// ---- VISUs/Home_Multidis2.TcVIS
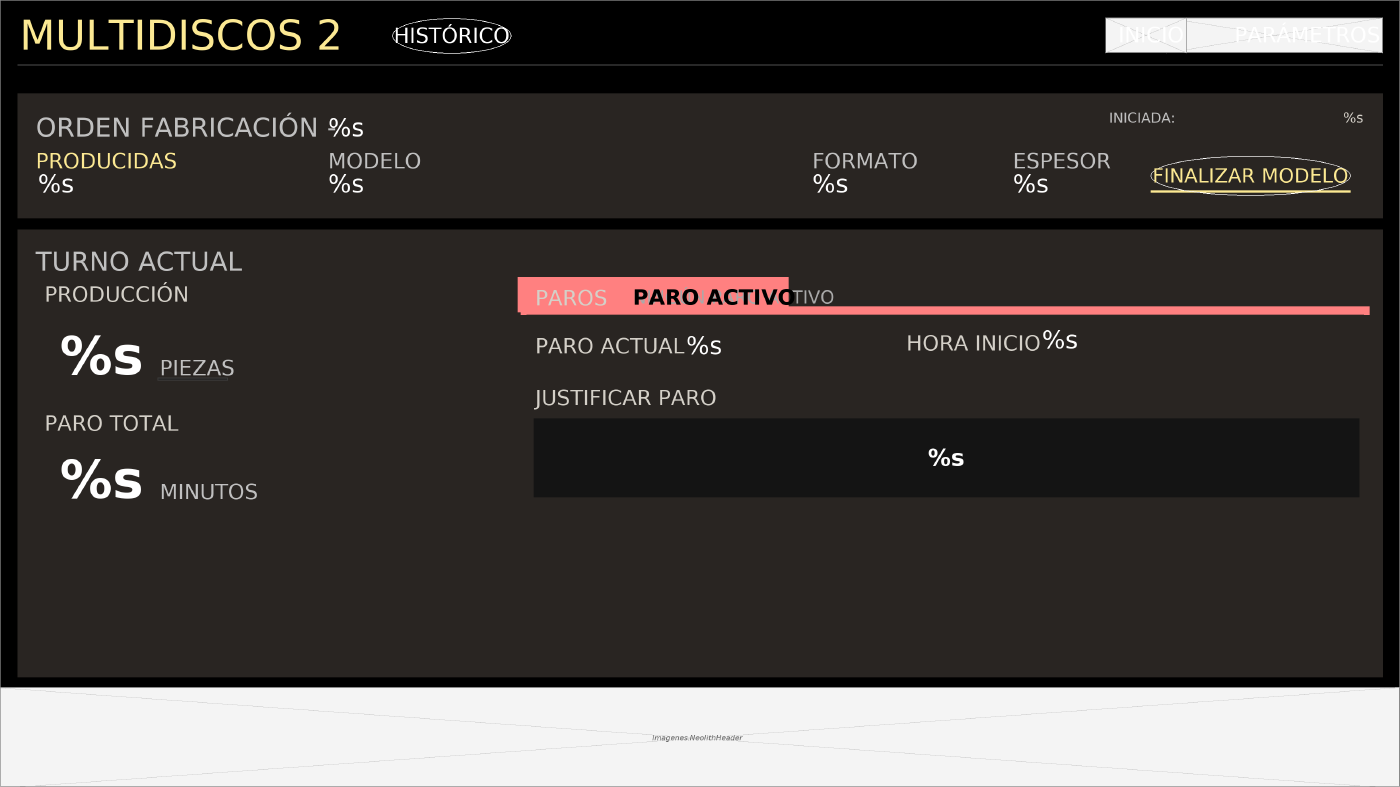
VISUALIZATION Home_Multidis2  // 1920x1080
    Ellipse (1479,1885 456x77), "Fin de producción del modelo"
        OnMouseClick: OpenDialog Dialog=V_Emerg_Fin_Prod_Md2, OpenModal=True, OpenCentered=True
    Lamp1 (869,1190 94x97), variable: FuncParoNodoMultidiscos.Funci_Multidiscos2.Fotocelula, style: Lamp-Lamp1-Yellow
    Rectangle (994,1445 183x30), "%s", text variable: FuncParoNodoCorteH4Remote1.Funci_CortHum4.H_InParo_Ftc, invisible if: FuncParoNodoMultidiscos.Funci_Multidiscos2.M_SinParo_Ftc
    Label (758,1444 239x30), "Hora Inicio del paro", invisible if: FuncParoNodoMultidiscos.Funci_Multidiscos2.M_SinParo_Ftc
    Rectangle (994,1503 192x30), "%s", text variable: FuncParoNodoCorteH4Remote1.Funci_CortHum4.Min_Parado_Ftc, invisible if: FuncParoNodoMultidiscos.Funci_Multidiscos2.M_SinParo_Ftc
    Label (793,1503 204x30), "Minutos Parado", invisible if: FuncParoNodoMultidiscos.Funci_Multidiscos2.M_SinParo_Ftc
    Label (753,1558 244x30), "Tiempo entre Piezas"
    Label (742,1594 255x62), "Tiempo entre Piezas Anterior"
    Rectangle (172,1318 183x123), "%s", text variable: FuncParoNodoMultidiscos.Funci_Multidiscos2.Cont_Piezas_Ftc
    Rectangle (994,1558 192x30), "%s", text variable: FuncParoNodoCorteH4Remote1.Funci_CortHum4.t_Entre_Piez_Ftc
    Rectangle (994,1610 192x30), "%s", text variable: FuncParoNodoCorteH4Remote1.Funci_CortHum4.t_Entr_Piez_Ante_Ftc
    Label (718,1127 397x30), "Sensor presencia tabla"
    Label (753,1348 326x30), "En producción todo OK", invisible if: FuncParoNodoMultidiscos.Funci_Multidiscos2.MParo_Ftc
    Label (571,1279 235x59), "Línea en paro", invisible if: FuncParoNodoMultidiscos.Funci_Multidiscos2.M_SinParo_Ftc
    Label (85,1180 361x144), "Número de losas"
    Label (1390,1230 361x56), "Modelo actual"
    Rectangle (1235,1324 671x53), "%s", text variable: FuncParoNodoMultidiscos.sModeloActualTabla_MD2
    Label (1390,1615 361x56), "Espesor"
    Rectangle (1235,1704 671x53), "%s", text variable: FuncParoNodoMultidiscos.sEspesorActualTabla_MD2
    Label (1390,1417 361x56), "Formato"
    Rectangle (1235,1506 671x53), "%s", text variable: FuncParoNodoMultidiscos.sFormatoActualTabla_MD2
    Rectangle (1533,1124 300x30), "%s", text variable: FuncParoNodoMultidiscos.sFechaInicModeloTab_MD2
    Label (1178,1125 354x30), "Fecha inicio del modelo actual"
    Rectangle (56,1801 1380x154), "%s", text variable: FuncParoNodoMultidiscos.Funci_Multidiscos2.S_Justi_Paro_Ftc, invisible if: FuncParoNodoMultidiscos.Funci_Multidiscos2.M_SinParo_Ftc
        OnMouseDown: write the text variable via Edit
    Label (55,1710 1381x106), "JUSTIFICAR EL PARO ACTUAL", invisible if: FuncParoNodoCorteH4Remote1.Funci_CortHum4.M_SinParo_Ftc
    Rectangle (24,315 1872x614)
    Rectangle (24,128 1872x171)
    Rectangle (24,88 1872x2)
    Label (24,16 514x64), "MULTIDISCOS 2"
    Rectangle (1426,451 183x30), "%s", text variable: FuncParoNodoCorteH4Remote1.Funci_CortHum4.H_InParo_Ftc, invisible if: FuncParoNodoMultidiscos.Funci_Multidiscos2.M_SinParo_Ftc
    Rectangle (938,459 192x30), "%s", text variable: FuncParoNodoCorteH4Remote1.Funci_CortHum4.Min_Parado_Ftc, invisible if: FuncParoNodoMultidiscos.Funci_Multidiscos2.M_SinParo_Ftc
    Label (46,148 390x54), "ORDEN FABRICACIÓN -"
    Rectangle (1573,147 300x30), "%s", text variable: FuncParoNodoMultidiscos.sFechaInicModeloTab_MD2
    Label (1518,147 99x30), "INICIADA:"
    Rectangle (732,574 1132x108), "%s", text variable: FuncParoNodoMultidiscos.Funci_Multidiscos2.S_Justi_Paro_Ftc, invisible if: FuncParoNodoMultidiscos.Funci_Multidiscos2.M_SinParo_Ftc
        OnMouseDown: write the text variable via Edit
    Image (1600,24 296x48), "PARÁMETROS"
        OnMouseClick: change screen: Ajustes_CorteH4
    Image (1516,24 111x48), "INICIO"
        OnMouseClick: change screen: Home_Sel_Maq
    Rectangle (447,232 671x40), "%s", text variable: FuncParoNodoMultidiscos.sModeloActualTabla_MD2
    Rectangle (1386,232 120x40), "%s", text variable: FuncParoNodoMultidiscos.sEspesorActualTabla_MD2
    Rectangle (1111,232 321x40), "%s", text variable: FuncParoNodoMultidiscos.sFormatoActualTabla_MD2
    Label (447,203 487x36), "MODELO"
    Label (1111,203 156x36), "FORMATO"
    Label (1386,203 156x36), "ESPESOR"
    Rectangle (447,155 321x40), "%s", text variable: FuncParoNodoCorteH4Remote1.sFormatoActualTabla
    Label (46,203 199x36), "PRODUCIDAS"
    Rectangle (49,232 248x40), "%s", text variable: FuncParoNodoCorteH4Remote1.sEspesorActualTabla
    Group (1578,214 274x54)
        Rectangle (0,47 274x3)
        Ellipse (0,0 274x54), "FINALIZAR MODELO"
            OnMouseClick: OpenDialog Dialog=V_Emerg_Fin_Prod_Md2, OpenModal=True, OpenCentered=True
    Label (46,332 390x54), "TURNO ACTUAL"
    Label (58,386 199x36), "PRODUCCIÓN"
    Label (731,457 261x36), "PARO ACTUAL", invisible if: FuncParoNodoMultidiscos.Funci_Multidiscos2.M_SinParo_Ftc
    Label (1240,453 261x36), "HORA INICIO", invisible if: FuncParoNodoMultidiscos.Funci_Multidiscos2.M_SinParo_Ftc
    Rectangle (79,444 183x88), "%s", text variable: FuncParoNodoMultidiscos.Funci_Multidiscos2.Cont_Piezas_Ftc
    Label (216,487 106x36), "PIEZAS"
    Rectangle (216,518 96x4), colour toggle: FuncParoNodoCorteH4Remote1.Funci_CortHum4.Fotocelula
    Label (731,528 261x36), "JUSTIFICAR PARO", invisible if: FuncParoNodoMultidiscos.Funci_Multidiscos2.M_SinParo_Ftc
    Rectangle (714,424 1164x4), invisible if: FuncParoNodoMultidiscos.Funci_Multidiscos2.M_SinParo_Ftc
    Rectangle (710,380 371x48), invisible if: FuncParoNodoMultidiscos.Funci_Multidiscos2.M_SinParo_Ftc
    Label (731,391 199x36), "PAROS"
    Label (865,393 326x30), "NINGÚN PARO ACTIVO", invisible if: FuncParoNodoMultidiscos.Funci_Multidiscos2.MParo_Ftc
    Label (865,393 235x30), "PARO ACTIVO", invisible if: FuncParoNodoMultidiscos.Funci_Multidiscos2.M_SinParo_Ftc
    Ellipse (538,25 163x48), "HISTÓRICO"
        OnMouseClick: change screen: HistTablaTablas_Ch4
    Label (58,563 261x36), "PARO TOTAL"
    Rectangle (79,614 183x88), "%s", text variable: FuncParoNodoCorteH4Remote1.Funci_CortHum4.Cont_Piezas_Ftc
    Label (216,657 142x36), "MINUTOS"
    Image (-7,943 1927x139), image: Imagenes.NeolithHeader
END_VISUALIZATION

// ---- VISUs/Listas_Para_Desplegables/FormatoTabla.TcTLO
TEXTLIST FormatoTabla
  0 = 'Sin seleccionar'
  1 = '170x170'
  2 = '200x650'
  3 = '300x150'
  4 = '300x300'
  5 = '30x30'
  6 = 'Ninguno de la lista'
   = ''
END_TEXTLIST

// ---- VISUs/Modelo_Tabla_Ch4.TcVIS
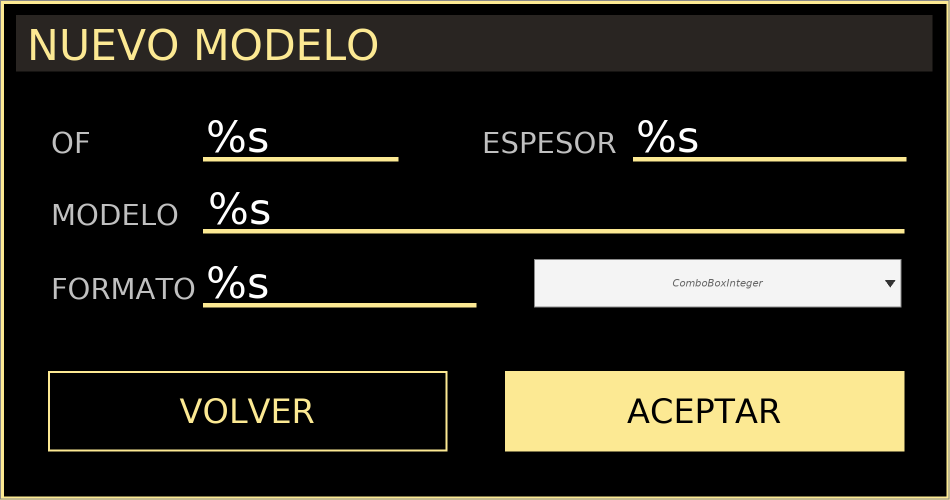
VISUALIZATION Modelo_Tabla_Ch4  // 950x500
    Rectangle (16,15 916x56)
    Rectangle (0,0 950x500)
    Label (24,17 498x56), "NUEVO MODELO"
    Rectangle (136,1125 690x58), "%s Contador piezas corte húmedo 4", text variable: FuncParoNodoCorteH4Remote1.CortHum4StrFuncParoEnviar.Cont_Piezas
    Button (871,1105 269x91), "Reset contador"
        tap FuncParoNodoCorteH4Remote1.Funci_CortHum4.ResetContPiez
    ComboBoxInteger (534,259 367x48), variable: FuncParoNodoCorteH4Remote1.FunGeneCortHum4.IndexListFormatoTabla, text list: 'FormatoTabla'
        p1601986498: ''
    Rectangle (205,185 701x48), "%s", text variable: FuncParoNodoCorteH4Remote1.FunGeneCortHum4.s_ModeloEleccionTabla
        OnMouseDown: write the text variable via Edit
    Label (48,197 148x36), "MODELO"
    Rectangle (203,229 701x4)
    Group (48,259 428x48), text variable: FuncParoNodoCorteH4Remote1.FunGeneCortHum4.s_FormatoEleccionTabla, input disabled if: FuncParoNodoCorteH4Remote1.FunGeneCortHum4.IndexListFormatoTabla<>0
        OnMouseClick: write the text variable via Edit
        Rectangle (155,0 273x48), "%s", text variable: FuncParoNodoCorteH4Remote1.sFormatoActualTabla
            OnMouseDown: write the text variable via Edit
        Label (0,12 148x36), "FORMATO"
        Rectangle (155,44 273x4)
    Group (479,113 427x48), "%s", text variable: FuncParoNodoCorteH4Remote1.FunGeneCortHum4.s_EspesorEleccionTabla
        OnMouseDown: write the text variable via Edit
        Rectangle (154,0 273x48), "%s", text variable: FuncParoNodoCorteH4Remote1.sEspesorActualTabla
            OnMouseDown: write the text variable via Edit
        Label (0,12 148x36), "ESPESOR"
        Rectangle (154,44 273x4)
    Rectangle (505,371 399x80), "ACEPTAR"
        tap FuncParoNodoCorteH4Remote1.FunGeneCortHum4.P_EscribirModelo
        OnMouseClick: CloseDialog Dialog=Modelo_Tabla_Ch4, Result=OK, NumpadKeypadSet=True
    Rectangle (48,371 399x80), "VOLVER"
        OnMouseClick: CloseDialog Dialog=Modelo_Tabla_Ch4, Result=Cancel, NumpadKeypadSet=True
    Group (48,113 350x48)
        Rectangle (155,0 195x48), "%s", text variable: FuncParoNodoCorteH4Remote1.sEspesorActualTabla
            OnMouseDown: write the text variable via Edit
        Label (0,12 148x36), "OF"
        Rectangle (155,44 195x4)
END_VISUALIZATION

// ---- VISUs/Ajustes_CorteH4.TcVIS
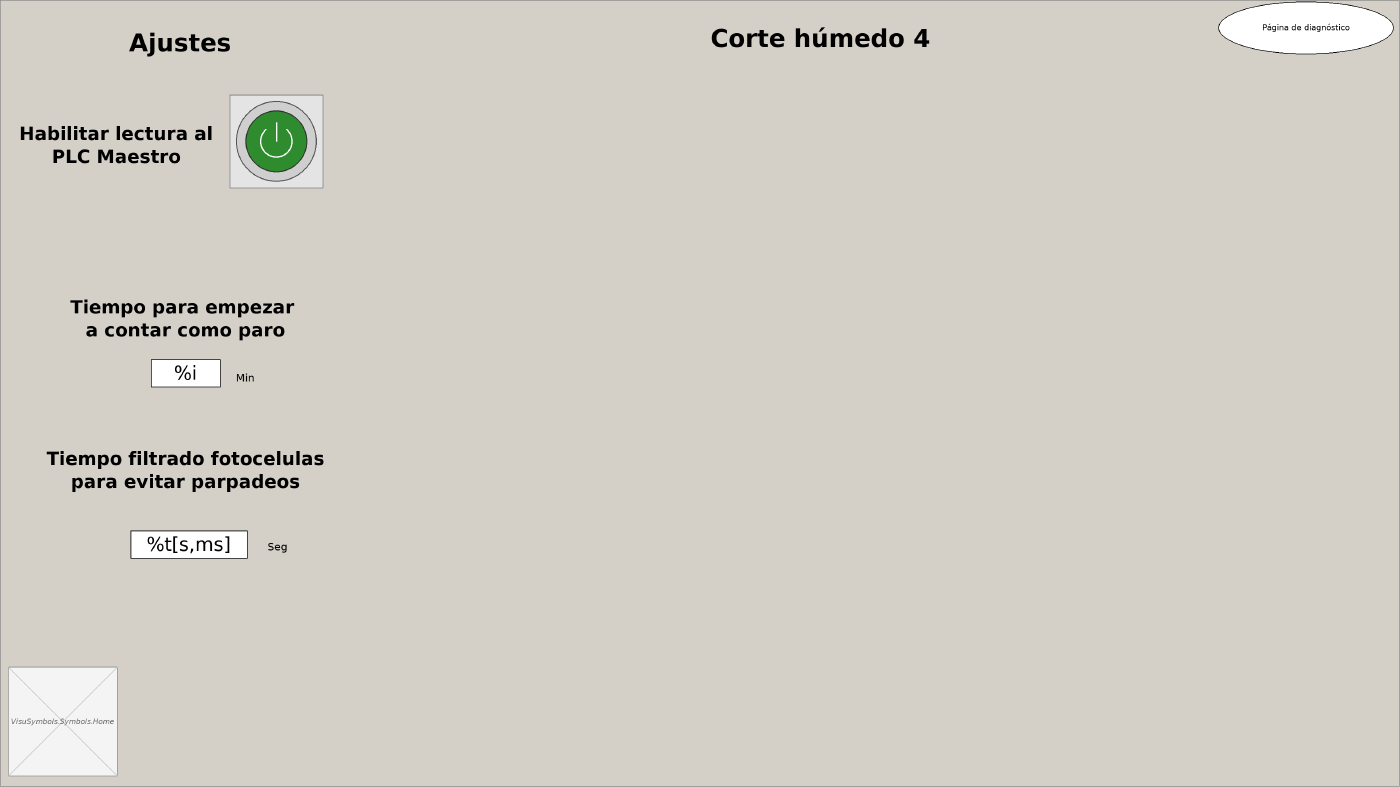
VISUALIZATION Ajustes_CorteH4  // 1920x1080
    Label (143,29 208x59), "Ajustes"
    Image (11,915 150x150), image: VisuSymbols.Symbols.Home
        OnMouseClick: change screen: Home_CortH4
    Label (22,144 275x110), "Habilitar lectura al PLC Maestro"
    PowerSwitch (315,128 128x132), variable: MAIN_Orden_Lectura_PLCs.bHabilitaLectura_Maestro, behaviour: TOGGLE, style: Switch-PowerSwitch-Green
    Label (82,390 345x94), "Tiempo para empezar a contar como paro"
    Label (160,482 188x30)
    Rectangle (207,493 95x38), "%i", text variable: FuncParoNodoCorteH4Remote1.HMI_Tiempo_Offset_MParo
        OnMouseDown: write the text variable via Edit
    Label (307,500 59x37), "Min"
    Label (58,598 393x94), "Tiempo filtrado fotocelulas para evitar parpadeos"
    Label (351,732 59x37), "Seg"
    Rectangle (179,728 160x38), "%t[s,ms]", text variable: FuncParoNodoCorteH4Remote1.HMI_TiempoFiltradoFotocel
        OnMouseDown: write the text variable via Edit
    Label (925,23 401x59), "Corte húmedo 4"
    Ellipse (1671,2 240x72), "Página de diagnóstico"
        OnMouseClick: change screen: DiagnosticoFB
END_VISUALIZATION

// ---- VISUs/Home_Sel_Maq.TcVIS
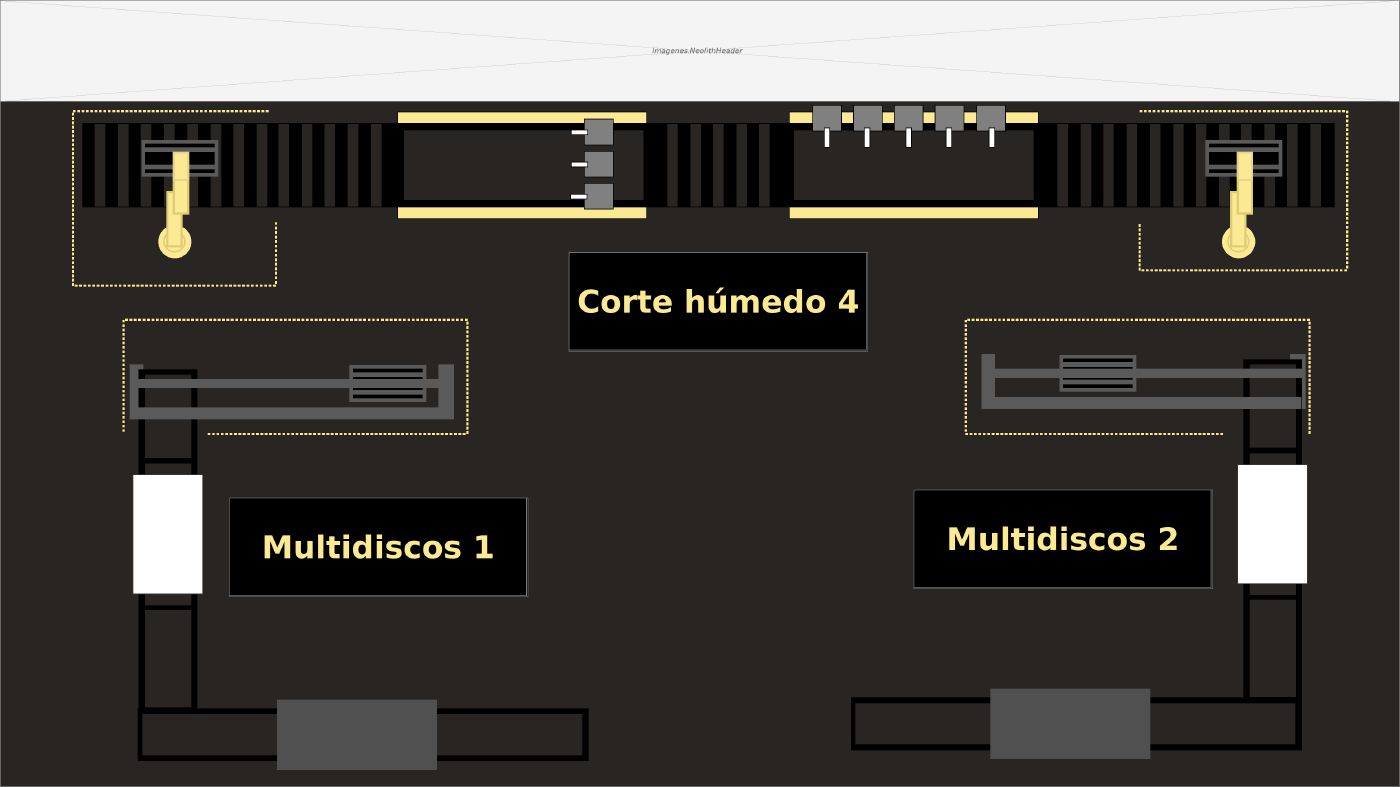
VISUALIZATION Home_Sel_Maq  // 1920x1080
    Button (780,346 410x136), "Corte húmedo 4"
        OnMouseUp: change screen: Home_CortH4
    Button (314,683 410x136), "Multidiscos 1"
        OnMouseUp: change screen: Home_Multidis1
    Button (1253,672 410x136), "Multidiscos 2"
        OnMouseDown: change screen: Home_Multidis2
    Image (-7,0 1927x139), image: Imagenes.NeolithHeader
    Group (100,144 1747x248)
        Rectangle (445,9 342x147)
        Rectangle (982,9 342x147)
        Rectangle (13,25 1717x115)
        Group (1349,25 363x115)
            Rectangle (0,0 16x115)
            Rectangle (32,0 16x115)
            Group (63,0 48x115)
                Rectangle (0,0 16x115)
                Rectangle (32,0 16x115)
            Group (127,0 111x115)
                Rectangle (0,0 16x115)
                Rectangle (32,0 16x115)
                Group (63,0 48x115)
                    Rectangle (0,0 16x115)
                    Rectangle (32,0 16x115)
            Rectangle (252,0 16x115)
            Rectangle (284,0 16x115)
            Group (315,0 48x115)
                Rectangle (0,0 16x115)
                Rectangle (32,0 16x115)
        Group (29,25 363x115)
            Rectangle (0,0 16x115)
            Rectangle (32,0 16x115)
            Group (63,0 48x115)
                Rectangle (0,0 16x115)
                Rectangle (32,0 16x115)
            Group (127,0 111x115)
                Rectangle (0,0 16x115)
                Rectangle (32,0 16x115)
                Group (63,0 48x115)
                    Rectangle (0,0 16x115)
                    Rectangle (32,0 16x115)
            Rectangle (252,0 16x115)
            Rectangle (284,0 16x115)
            Group (315,0 48x115)
                Rectangle (0,0 16x115)
                Rectangle (32,0 16x115)
        Rectangle (408,25 16x115)
        Rectangle (453,34 330x97)
        Rectangle (701,19 40x36)
        Rectangle (701,63 40x36)
        Rectangle (701,107 40x36)
        Rectangle (683,34 23x7)
        Rectangle (683,78 23x7)
        Rectangle (682,122 23x7)
        Rectangle (988,34 330x97)
        Rectangle (1014,0 40x36)
        Rectangle (1070,0 40x36)
        Rectangle (1126,0 40x36)
        Rectangle (1182,0 40x36)
        Rectangle (1239,0 40x36)
        Rectangle (1085,31 8x27)
        Rectangle (1030,31 8x27)
        Rectangle (1142,31 8x27)
        Rectangle (1197,31 8x27)
        Rectangle (1256,31 8x27)
        Group (814,25 142x115)
            Rectangle (126,0 16x115)
            Rectangle (0,0 16x115)
            Rectangle (32,0 16x115)
            Group (63,0 48x115)
                Rectangle (0,0 16x115)
                Rectangle (32,0 16x115)
        Polyline (1463,8) (1747,8) (1747,227) (1463,227) (1463,161)
        Polyline (278,161) (278,248) (0,248) (0,8) (271,8)
        Group (94,48 105x162)
            Ellipse (23,117 45x45)
            Ellipse (30,124 30x30)
            RoundedRectangle (34,70 22x77)
            RoundedRectangle (0,0 105x50)
            Rectangle (0,10 105x6)
            Rectangle (0,34 105x6)
            RoundedRectangle (43,25 22x77)
            RoundedRectangle (43,16 22x40)
        Group (1553,48 105x162)
            Ellipse (23,117 45x45)
            Ellipse (30,124 30x30)
            RoundedRectangle (34,70 22x77)
            RoundedRectangle (0,0 105x50)
            Rectangle (0,10 105x6)
            Rectangle (0,34 105x6)
            RoundedRectangle (43,25 22x77)
            RoundedRectangle (43,16 22x40)
    Group (1167,439 629x602)
        Rectangle (544,362 65x16)
        Rectangle (0,518 618x72)
        Polyline (629,156) (629,0) (157,0) (157,156) (513,156)
        Group (286,48 57x50)
            RoundedRectangle (0,0 105x50)
            Rectangle (0,10 105x6)
            Rectangle (0,34 105x6)
        Rectangle (602,47 21x75)
        Rectangle (179,47 18x75)
        Rectangle (538,54 80x465)
        Rectangle (546,60 65x116)
        Rectangle (546,182 65x196)
        Rectangle (530,198 96x164)
        Rectangle (546,383 65x135)
        Rectangle (5,525 605x58)
        Rectangle (191,506 219x96)
        Rectangle (193,106 424x16)
        Rectangle (190,67 431x12)
    Group (169,439 638x617)
        Rectangle (20,533 618x72)
        Polyline (116,156) (472,156) (472,0) (0,0) (0,156)
        Group (310,62 57x50)
            RoundedRectangle (0,0 105x50)
            Rectangle (0,10 105x6)
            Rectangle (0,34 105x6)
        Rectangle (432,61 21x75)
        Rectangle (9,61 18x75)
        Rectangle (21,68 80x465)
        Rectangle (29,74 65x116)
        Rectangle (29,196 65x196)
        Rectangle (13,212 96x164)
        Rectangle (29,397 65x135)
        Rectangle (25,540 605x58)
        Rectangle (211,521 219x96)
        Rectangle (17,120 430x16)
        Rectangle (20,81 431x12)
END_VISUALIZATION

// ---- VISUs/HistTablaTablas_Ch4.TcVIS
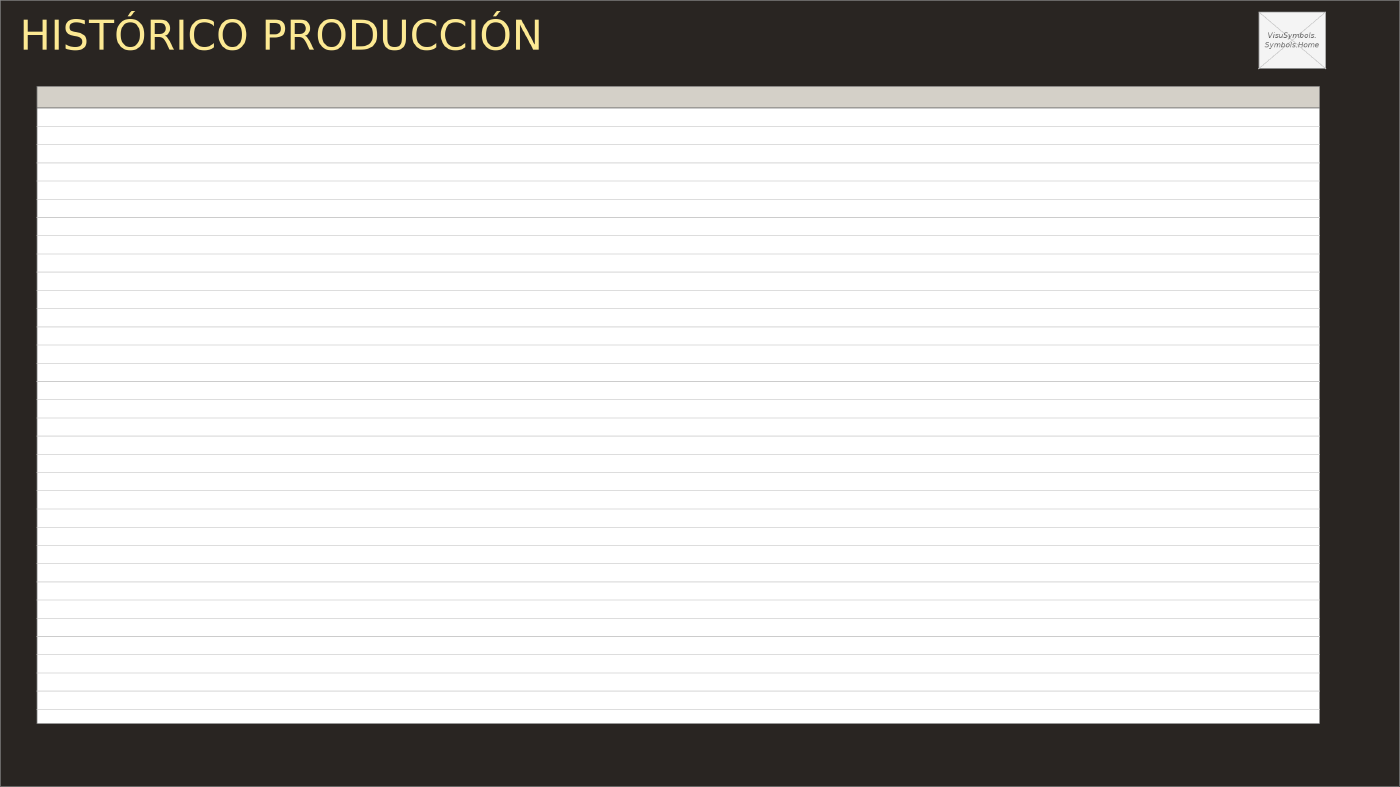
VISUALIZATION HistTablaTablas_Ch4  // 1920x1080
    Image (1726,16 92x78), image: VisuSymbols.Symbols.Home
        OnMouseClick: change screen: Home_CortH4
    Table (50,118 1760x875), data array: RegistroLocalDataBase.aHistoricStrTablasCH4
        p3854506369: RegistroLocalDataBase.aHistoricStrTablasCH4[INDEX].ID
        p1892666644: RegistroLocalDataBase.aHistoricStrTablasCH4[INDEX].Fecha
        p338671338: RegistroLocalDataBase.aHistoricStrTablasCH4[INDEX].Modelo
        p2170511999: RegistroLocalDataBase.aHistoricStrTablasCH4[INDEX].Formato
        p3723444502: RegistroLocalDataBase.aHistoricStrTablasCH4[INDEX].Espesor
        p1218418051: RegistroLocalDataBase.aHistoricStrTablasCH4[INDEX].Maquina
        p746581629: RegistroLocalDataBase.aHistoricStrTablasCH4[INDEX].Cont_Piezas
        p3104783080: RegistroLocalDataBase.aHistoricStrTablasCH4[INDEX].t_Entre_Piez_Ftc
        p2501879983: RegistroLocalDataBase.aHistoricStrTablasCH4[INDEX].S_Justi_Paro_Ftc
        p1757482276: Numero de tablas
        p4088588272: Tiempo entre tablas
        p2243050616: Justif paro
    Label (24,16 669x64), "HISTÓRICO PRODUCCIÓN"
END_VISUALIZATION

// ---- VISUs/Modelo_Tabla_Md1.TcVIS
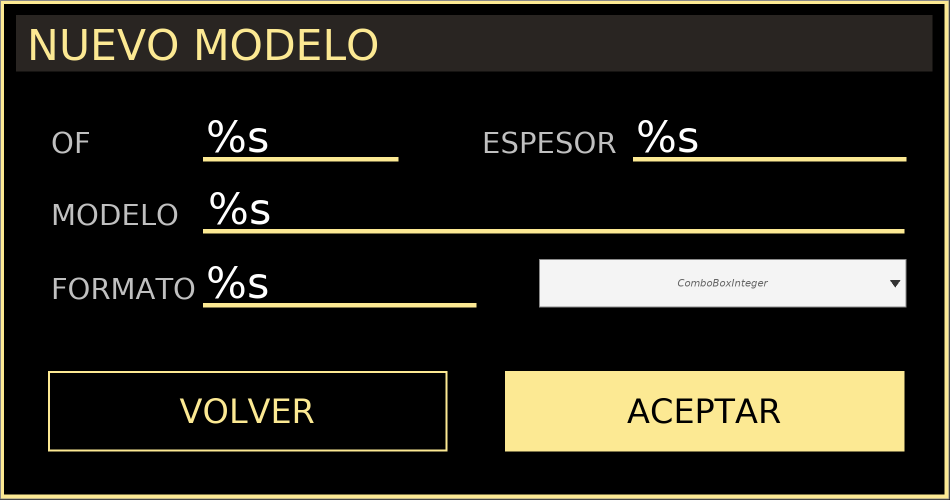
VISUALIZATION Modelo_Tabla_Md1  // 950x500
    Rectangle (28,569 690x58), "%s Contador piezas Multidiscos 1", text variable: FuncParoNodoMultidiscos.Funci_Multidiscos1.Cont_Piezas_Ftc
    Button (763,549 269x91), "Reset contador"
        tap FuncParoNodoMultidiscos.Funci_Multidiscos1.Pul_Reset_Cnt_Piez
    ComboBoxInteger (539,259 367x48), variable: FuncParoNodoMultidiscos.FunGeneMultidiscos1.IndexListFormatoTabla, text list: 'FormatoTabla'
    Rectangle (16,15 916x56)
    Rectangle (0,0 948x498)
    Label (24,17 498x56), "NUEVO MODELO"
    Rectangle (205,185 701x48), "%s", text variable: FuncParoNodoMultidiscos.FunGeneMultidiscos1.s_ModeloEleccionTabla
        OnMouseDown: write the text variable via Edit
    Label (48,197 148x36), "MODELO"
    Rectangle (203,229 701x4)
    Rectangle (203,259 273x48), "%s", text variable: FuncParoNodoMultidiscos.FunGeneMultidiscos1.s_FormatoEleccionTabla, input disabled if: FuncParoNodoMultidiscos.FunGeneMultidiscos1.IndexListFormatoTabla<>0
        OnMouseDown: write the text variable via Edit
    Label (48,271 148x36), "FORMATO"
    Rectangle (203,303 273x4)
    Rectangle (633,113 273x48), "%s", text variable: FuncParoNodoMultidiscos.FunGeneMultidiscos1.s_EspesorEleccionTabla
        OnMouseDown: write the text variable via Edit
    Label (479,125 148x36), "ESPESOR"
    Rectangle (633,157 273x4)
    Rectangle (505,371 399x80), "ACEPTAR"
        tap FuncParoNodoMultidiscos.FunGeneMultidiscos1.P_EscribirModelo
        OnMouseClick: CloseDialog Dialog=Modelo_Tabla_Md1, Result=OK, NumpadKeypadSet=True
    Rectangle (48,371 399x80), "VOLVER"
        OnMouseClick: CloseDialog Dialog=Modelo_Tabla_Md1, Result=Cancel, NumpadKeypadSet=True
    Group (48,113 350x48)
        Rectangle (155,0 195x48), "%s", text variable: FuncParoNodoCorteH4Remote1.sEspesorActualTabla
            OnMouseDown: write the text variable via Edit
        Label (0,12 148x36), "OF"
        Rectangle (155,44 195x4)
END_VISUALIZATION

// ---- VISUs/Modelo_Tabla_Md2.TcVIS
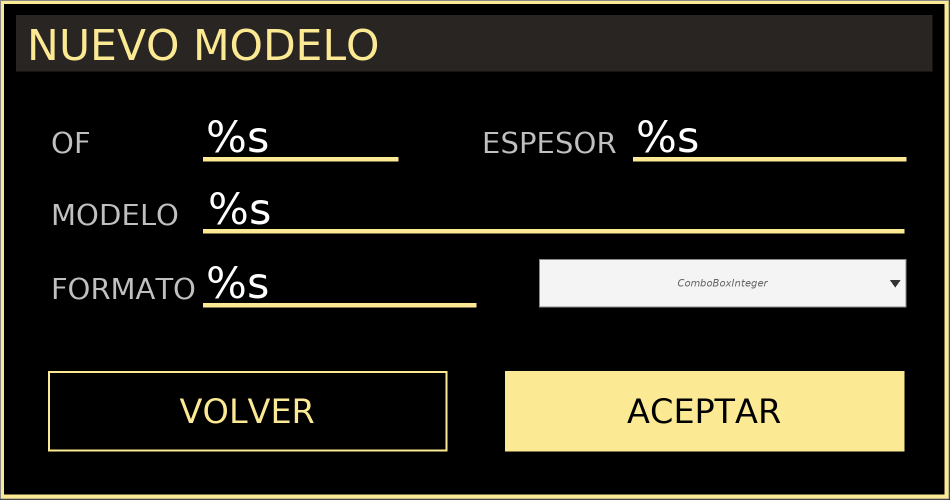
VISUALIZATION Modelo_Tabla_Md2  // 950x500
    Rectangle (0,0 948x498)
    Rectangle (424,1281 690x58), "%s Contador piezas Multidiscos 2", text variable: FuncParoNodoMultidiscos.Funci_Multidiscos2.Cont_Piezas_Ftc
    Button (1159,1261 269x91), "Reset contador"
        tap FuncParoNodoMultidiscos.Funci_Multidiscos2.Pul_Reset_Cnt_Piez
    ComboBoxInteger (539,259 367x48), variable: FuncParoNodoMultidiscos.FunGeneMultidiscos2.IndexListFormatoTabla, text list: 'FormatoTabla'
    Rectangle (16,15 916x56)
    Label (24,17 498x56), "NUEVO MODELO"
    Rectangle (205,185 701x48), "%s", text variable: FuncParoNodoMultidiscos.FunGeneMultidiscos2.s_ModeloEleccionTabla
        OnMouseDown: write the text variable via Edit
    Label (48,197 148x36), "MODELO"
    Rectangle (203,229 701x4)
    Rectangle (203,259 273x48), "%s", text variable: FuncParoNodoMultidiscos.FunGeneMultidiscos2.s_FormatoEleccionTabla, input disabled if: FuncParoNodoMultidiscos.FunGeneMultidiscos2.IndexListFormatoTabla<>0
        OnMouseDown: write the text variable via Edit
    Label (48,271 148x36), "FORMATO"
    Rectangle (203,303 273x4)
    Rectangle (633,113 273x48), "%s", text variable: FuncParoNodoMultidiscos.FunGeneMultidiscos2.s_EspesorEleccionTabla
        OnMouseDown: write the text variable via Edit
    Label (479,125 148x36), "ESPESOR"
    Rectangle (633,157 273x4)
    Rectangle (505,371 399x80), "ACEPTAR"
        tap FuncParoNodoMultidiscos.FunGeneMultidiscos2.P_EscribirModelo
        OnMouseClick: CloseDialog Dialog=Modelo_Tabla_Md2, Result=OK, NumpadKeypadSet=True
    Rectangle (48,371 399x80), "VOLVER"
        OnMouseClick: CloseDialog Dialog=Modelo_Tabla_Md2, Result=Cancel, NumpadKeypadSet=True
    Group (48,113 350x48)
        Rectangle (155,0 195x48), "%s", text variable: FuncParoNodoCorteH4Remote1.sEspesorActualTabla
            OnMouseDown: write the text variable via Edit
        Label (0,12 148x36), "OF"
        Rectangle (155,44 195x4)
END_VISUALIZATION

// ---- VISUs/V_Emerg_Fin_Prod_Ch4.TcVIS
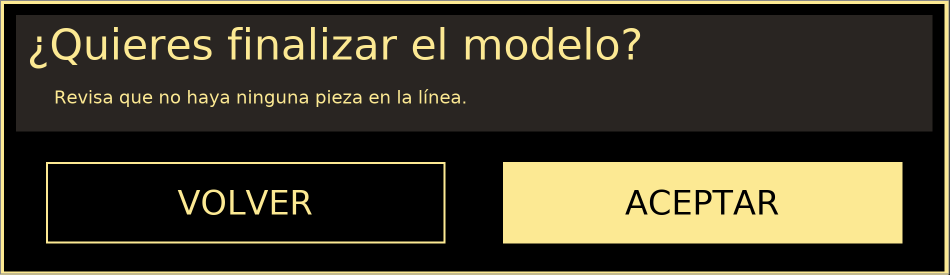
VISUALIZATION V_Emerg_Fin_Prod_Ch4  // 950x275
    Rectangle (0,0 948x275)
    Rectangle (16,15 916x116)
    Label (24,17 898x65), "¿Quieres finalizar el modelo?"
    Label (51,85 857x43), "Revisa que no haya ninguna pieza en la línea."
    Rectangle (503,162 399x81), "ACEPTAR"
        tap FuncParoNodoCorteH4Remote1.FunGeneCortHum4.P_FinProduccion
        OnMouseClick: CloseDialog Dialog=V_Emerg_Fin_Prod_Ch4, Result=OK, NumpadKeypadSet=True
        OnMouseClick: OpenDialog Dialog=Modelo_Tabla_Ch4, OpenModal=True, OpenCentered=True
    Rectangle (46,162 399x81), "VOLVER"
        OnMouseClick: CloseDialog Dialog=V_Emerg_Fin_Prod_Ch4, Result=Cancel, NumpadKeypadSet=True
END_VISUALIZATION

// ---- VISUs/V_Emerg_Fin_Prod_Md2.TcVIS
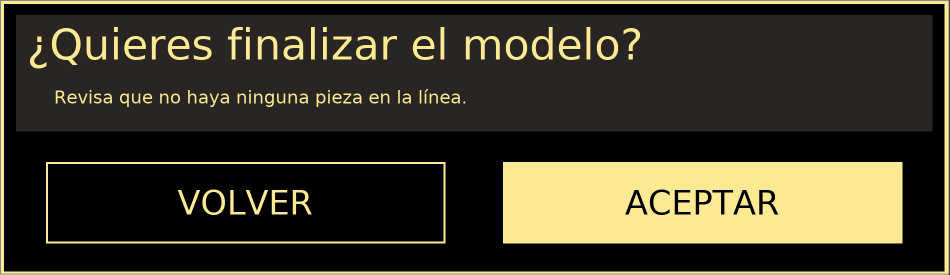
VISUALIZATION V_Emerg_Fin_Prod_Md2  // 950x275
    Rectangle (0,0 948x275)
    Rectangle (16,15 916x116)
    Label (24,17 898x65), "¿Quieres finalizar el modelo?"
    Label (51,85 857x43), "Revisa que no haya ninguna pieza en la línea."
    Rectangle (503,162 399x81), "ACEPTAR", text variable: FuncParoNodoMultidiscos.FunGeneMultidiscos2.P_FinProduccion
        tap FuncParoNodoMultidiscos.FunGeneMultidiscos2.P_FinProduccion
        OnMouseClick: CloseDialog Dialog=V_Emerg_Fin_Prod_Md2, Result=OK, NumpadKeypadSet=True
        OnMouseClick: OpenDialog Dialog=Modelo_Tabla_Md2, OpenModal=True, OpenCentered=True
    Rectangle (46,162 399x81), "VOLVER"
        OnMouseClick: CloseDialog Dialog=V_Emerg_Fin_Prod_Md2, Result=Cancel, NumpadKeypadSet=True
END_VISUALIZATION

// ---- VISUs/V_Emerg_Fin_Prod_Md1.TcVIS
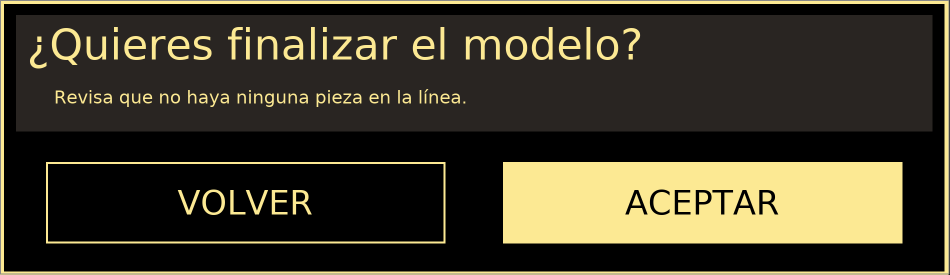
VISUALIZATION V_Emerg_Fin_Prod_Md1  // 950x275
    Rectangle (0,0 948x275)
    Rectangle (16,15 916x116)
    Label (24,17 898x65), "¿Quieres finalizar el modelo?"
    Label (51,85 857x43), "Revisa que no haya ninguna pieza en la línea."
    Rectangle (503,162 399x81), "ACEPTAR"
        tap FuncParoNodoMultidiscos.FunGeneMultidiscos1.P_FinProduccion
        OnMouseClick: CloseDialog Dialog=V_Emerg_Fin_Prod_Md1, Result=OK, NumpadKeypadSet=True
        OnMouseClick: OpenDialog Dialog=Modelo_Tabla_Md1, OpenModal=True, OpenCentered=True
    Rectangle (46,162 399x81), "VOLVER"
        OnMouseClick: CloseDialog Dialog=V_Emerg_Fin_Prod_Md1, Result=Cancel, NumpadKeypadSet=True
END_VISUALIZATION
